Universal Robots PolyScope program: a.urp

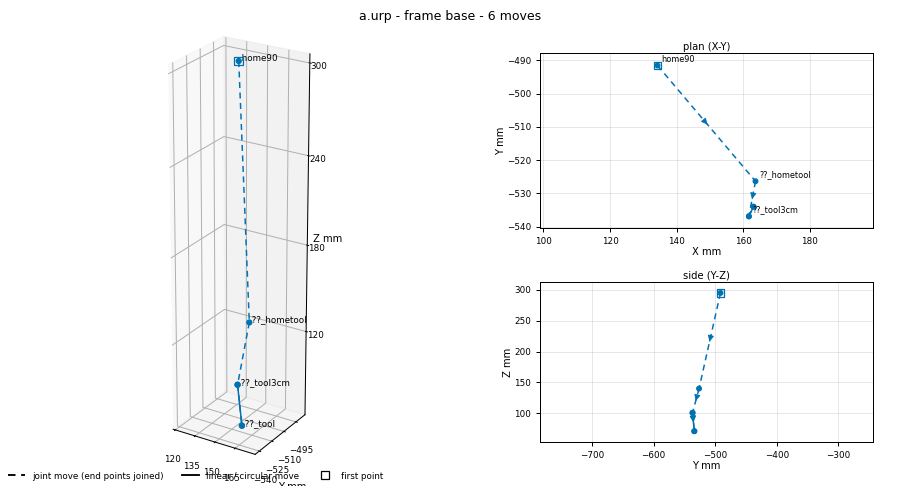
[picture p0: tool path of a.urp in frame base, 6 of 7 moves have a stored position in this frame; points joined in program order, loops and branches not executed]
Program a (installation=20240827 directory=/programs/Demos/0208 createdIn=5.15.1 lastSavedIn=5.15.1 robotSerialNumber=20245500285)
Calibrated DH parameters: a=[0.000097, -0.210459, -0.026602, 0.000137, 0.000078, 0]; d=[0.162601, 254.180657, -54.076236, -199.970743, 0.099615, 0.099684]; alpha=[1.569796, -0.001455, 0.001957, 1.570525, -1.571561, 0]; deltaTheta=[0, -1.053331, 8.839472, -1.50296, 0.000002, 0]
InitVariablesNode
Robot Program (runOnlyOnce=true)
  MoveJ speed 60 deg/s, acceleration 80 deg/s^2 (useActiveTCP=true) feature=Base
    Waypoint home90: TCP in base x=134.286 y=-491.541 z=295.223 mm, rx=-2.2176 ry=-2.2241 rz=-0.0004 rad; joints [90, -90, 90, -90, -90, 90] deg; TCP offset x=-0.17 y=0 z=192.95 mm, rx=0 ry=0 rz=0 rad
    Waypoint 路点_hometool: TCP in base x=163.745 y=-526.322 z=139.992 mm, rx=-2.2176 ry=-2.2241 rz=-0.0004 rad; joints [93.175, -80.187, 102.521, -112.33, -90.048, 93.18] deg; TCP offset x=-0.17 y=0 z=192.95 mm, rx=0 ry=0 rz=0 rad
    Waypoint 路点_tool3cm: TCP in base x=161.75 y=-536.883 z=100.635 mm, rx=-2.2176 ry=-2.2241 rz=-0.0004 rad; joints [92.902, -76.645, 104.479, -117.832, -90.062, 92.907] deg
    Waypoint 路点_tool: TCP in base x=163.14 y=-533.982 z=70.738 mm, rx=-2.2176 ry=-2.2241 rz=-0.0004 rad; joints [93.064, -74.843, 107.171, -122.327, -90.072, 93.069] deg
    SuppressedNode
      Popup Message (haltProgram=false message=3cm inputType=Text)
    poseget := 路点_toolget_actual_tcp_pose()
    zz3cm := p[0,0,0.03,0,0,0]
    pose := pose_add(路点_tool, zz3cm)
    Waypoint Variable (Variable): variable=pose
    MoveL speed 50 mm/s, acceleration 500 mm/s^2 (useActiveTCP=true) feature=Base
      Waypoint 路点_tool3cm: TCP in base x=161.75 y=-536.883 z=100.635 mm, rx=-2.2176 ry=-2.2241 rz=-0.0004 rad; joints [92.902, -76.645, 104.479, -117.832, -90.062, 92.907] deg
      Wait Sleep waitTime=1
    MoveL speed 250 mm/s, acceleration 1200 mm/s^2 (useActiveTCP=true) feature=Base
      Waypoint 路点_tool: TCP in base x=163.14 y=-533.982 z=70.738 mm, rx=-2.2176 ry=-2.2241 rz=-0.0004 rad; joints [93.064, -74.843, 107.171, -122.327, -90.072, 93.069] deg
